{attribute 'linkalways'} 
{attribute 'no_explicit_call' := 'This FB is a CLASS and must be accessed using methods or properties'}
{attribute 'enable_dynamic_creation'}
FUNCTION_BLOCK PUBLIC BasicDigitalInput IMPLEMENTS I_DigitalInput
VAR
	input AT %Q* : BOOL;
	inverted : BOOL;
END_VAR

METHOD FB_init : BOOL
VAR_INPUT
	bInitRetains : BOOL; // if TRUE, the retain variables are initialized (warm start / cold start)
	bInCopyCode : BOOL;  // if TRUE, the instance afterwards gets moved into the copy code (online change)
	inverted : BOOL;
END_VAR
THIS^.inverted := inverted;
END_METHOD

{attribute 'monitoring' := 'call'}
PROPERTY PUBLIC State : BOOL
GET // PUBLIC
State := input XOR inverted;
END_GET
END_PROPERTY

END_FUNCTION_BLOCK

(* stored: Version 1.1.0.1, ProductVersion 3.1.4024.12
   POU BasicDigitalInput: Id {4daa4205-83ad-4e31-b94b-9e2e1a1349e4}, SpecialFunc None
   Method FB_init: Id {3850ab49-bb61-42ea-ad81-8c5a8b891ffd}
   Property State: Id {33977c33-f3a3-4aeb-b136-a5b0f232dd15}
   Get Get: Id {405cd970-3f2e-4b9f-8a84-3f181dbee17e} *)
